// TwinCAT 3 PLC project Main
// ProgramVersion: 3.1.4023.0
// libraries:
//   Tc2_Standard, * (Beckhoff Automation GmbH)
//   Tc2_System, * (Beckhoff Automation GmbH)
//   Tc3_JsonXml, * (Beckhoff Automation GmbH)
//   Tc3_Module, * (Beckhoff Automation GmbH)
// project tree:
//   DUTs/ MyExampleInternalStructure.TcDUT, MyExampleStructure.TcDUT
//   / PlcTask.TcTTO
//   POUs/ MAIN.TcPOU
// real-time tasks:
//   TASK PlcTask: cycle T#10ms, priority 20, ADS port 350

CONFIGURATION Main
    RESOURCE PLC ON TwinCAT3
        TASK PlcTask(INTERVAL := T#10ms, PRIORITY := 20);
        PROGRAM MAIN WITH PlcTask : MAIN;
    END_RESOURCE
END_CONFIGURATION

// ---- DUTs/MyExampleInternalStructure.TcDUT
TYPE MyExampleInternalStructure :
STRUCT
	myUdint : UDINT := 999;
END_STRUCT
END_TYPE

// ---- DUTs/MyExampleStructure.TcDUT
TYPE MyExampleStructure :
STRUCT
	myInt : INT := 123;
	myBool : BOOL := TRUE;
	myString : STRING := 'hello';
	myArray : ARRAY[0..1] OF BYTE := [0, 255];
	myInternalStructure : MyExampleInternalStructure;
END_STRUCT
END_TYPE

// ---- POUs/MAIN.TcPOU
PROGRAM MAIN
VAR
	
	// variables used for testing.
	testVariable : MyExampleStructure;	
	
	// fb's needed. (You need to add TC3_XmlJson library in your references)
	transform : FB_JsonReadWriteDataType;
	
	(* datatype name (this is useful to ask TwinCAT what the structure is called, as it prevents
	   you from hard coding the name in your code.  Plus it continues to work if placed in a 
	   library, as all structures gain the library namespace. *)
	
	datatypeName : STRING(100); // this needs to be big enough to take the full structure name
	resultingJsonStringLength : UDINT; // not needed, but from this you can see how long the string will be. 
	jsonString : STRING(1000); // this is the destination of the json

END_VAR


(* first we get the datatype name of the structure / variable.  We could hard code this, but hard coding structure
   names in your code is not good practice, just in case you rename your structures later *)

datatypeName := transform.GetDataTypeNameByAddress(SIZEOF(testVariable),ADR(testVariable));

(* next we find out how big the resulting json string will be.  In the next step you will need a string of at least
   this big to fit the json in. *)

resultingJsonStringLength := transform.GetSizeJsonStringFromSymbol(datatypeName,SIZEOF(testVariable),ADR(testVariable));

(* finally the transformation step.  This requires the datatype name, the size and address of the source, and the size
   and address of the destination *)

transform.CopyJsonStringFromSymbol(datatypeName,SIZEOF(testVariable), ADR(testVariable),jsonString,SIZEOF(jsonString));

END_PROGRAM
